(* IEC 61131-3 sources: pub-control-lib/src/02_PubControl, 4 files *)

(* ---- Types.st ---- *)
NAMESPACE Siemens.PubControl.Types
    TYPE
        TankStatus : INT (ACTIVE := 0,  Tapped := 1, TANKING := 2, EMPTY := 4, SERVICE := 3) := ACTIVE;
    END_TYPE

    TYPE
        QualityData : STRUCT
            /// Time how long is tank full with medium (in days)
            occupancyPeriod : REAL;
            /// Time how long tank is empty (in days)
            emptinessPeriod : REAL;
            /// Time how long it needed to empty tank (in days)
            emptyingPeriod : REAL;
            /// delivery date
            deliveryDate : DATE_AND_TIME;
            /// Change inliner last time
            inlinerDate : DATE_AND_TIME;
        END_STRUCT;
    END_TYPE

END_NAMESPACE

(* ---- BasicTapBar.st ---- *)
USING Siemens.PubControl.Interfaces;

NAMESPACE Siemens.PubControl.TapBars
    CLASS BasicTapBar IMPLEMENTS ITapBar
        VAR PRIVATE
            consumption : REAL;
            lastConsumption : REAL;
            flow : REAL;
        END_VAR

        VAR PUBLIC
            WatchDogDiffTime : LTIME;
        END_VAR

        METHOD PUBLIC CalcImpulses
            VAR_INPUT
                MeasureTime : LTIME;
                Impulses : INT;
                Factor : INT;
            END_VAR
            VAR CONSTANT
                HOUR_IN_NS : REAL := REAL#3.6e12;
                ML_IN_L : REAL := REAL#1000.0;
            END_VAR
            VAR_TEMP
                calculatedTime : REAL := REAL#0.0;
            END_VAR
            lastConsumption := (Impulses * Factor)/ML_IN_L;
            consumption := consumption + lastConsumption;

            IF (LTIME#0ns < MeasureTime AND  MeasureTime < WatchDogDiffTime) THEN
                calculatedTime := (TO_REAL(TO_LINT(MeasureTime)));
                flow := lastConsumption * (HOUR_IN_NS/calculatedTime);
            END_IF;
        END_METHOD

        METHOD PUBLIC GetConsumption : REAL
            GetConsumption := consumption;
        END_METHOD

        METHOD PUBLIC GetFlow : REAL
            GetFlow := flow;
        END_METHOD

        METHOD PUBLIC Reset
            consumption := REAL#0.0;
            flow := REAL#0.0;
        END_METHOD

    END_CLASS
END_NAMESPACE

(* ---- TankTap.st ---- *)
USING Siemens.PubControl.Types;
USING Siemens.PubControl.Interfaces;
USING Siemens.PubControl.Types;

NAMESPACE Siemens.PubControl

    // TODO HMI Interface
    CLASS TankTap
        IMPLEMENTS ITank
        VAR PUBLIC
        END_VAR
        VAR PROTECTED
            _maxLevel : UINT;
            _status : TankStatus := TankStatus#ACTIVE;
            _currentLevel : REAL;
            _inTanking : BOOL;
            _inService : BOOL;
        END_VAR

        METHOD PUBLIC SetMaxLevel : INT
            VAR_INPUT
                /// Max level in liter
                MaxLevel : UINT;
            END_VAR
            IF MaxLevel > UINT#0 THEN
                _maxLevel := MaxLevel;
                SetMaxLevel := 0;
            ELSE
                SetMaxLevel := -1;
            END_IF;
            THIS.CheckStatus();
        END_METHOD
        // TODO Test me

        METHOD PUBLIC FINAL Consume : TankStatus
            VAR_INPUT
                /// consumption in liter
                consumption : REAL;
            END_VAR
            IF (_currentLevel - consumption) < 0 THEN
                _currentLevel := 0;
            ELSE
                _currentLevel := _currentLevel - consumption;
            END_IF;
            THIS.CheckStatus();
            Consume := _status;
        END_METHOD
        /// Level in liter

        METHOD PUBLIC GetLevel : UINT
            GetLevel := TO_UINT(_currentLevel);
        END_METHOD

        METHOD PUBLIC GetStatus : TankStatus
            THIS.CheckStatus();
            GetStatus := _status;
        END_METHOD

        METHOD PUBLIC Cleaning
            VAR_INPUT
                Start : BOOL;
                Stop : BOOL;
            END_VAR
            ;
        END_METHOD

        METHOD PROTECTED CheckStatus
            VAR_TEMP
                level : UINT;
            END_VAR
            level := TO_UINT(_currentLevel);
            IF UINT#0 < level AND level < _maxLevel THEN
                _status := TankStatus#TAPPED;
            ELSIF level <= UINT#0 THEN
                _status := TankStatus#EMPTY;
            ELSIF _inTanking THEN
                _status := TankStatus#TANKING;
            ELSIF _inService THEN
                _status := TankStatus#Service;
            ELSE
                _status := TankStatus#ACTIVE;
            END_IF;
        END_METHOD

        METHOD PUBLIC Tanking
            _inTanking := TRUE;
            _currentLevel := _maxLevel;
            _inTanking := FALSE;
        END_METHOD
    END_CLASS

END_NAMESPACE

(* ---- TankWeight.st ---- *)
USING Siemens.PubControl.Interfaces;
USING Siemens.PubControl.Types;

NAMESPACE Siemens.PubControl

    CLASS TankWeight EXTENDS TankTap
        VAR PUBLIC
            /// Weight in kilogram
            Weight : REAL;
        END_VAR
        VAR PROTECTED
            _maxLevelWeight : REAL;
            _factorLevelWeight : REAL;
        END_VAR

        METHOD PUBLIC OVERRIDE SetMaxLevel : INT
            VAR_INPUT
                /// Max level in liter
                MaxLevel : UINT;
            END_VAR
            IF Weight > 0 AND MaxLevel > UINT#0 THEN
                _maxLevel := MaxLevel;
                _currentLevel := MaxLevel;
                _maxLevelWeight := Weight;
                _factorLevelWeight := _maxLevel / _maxLevelWeight;
                SetMaxLevel := 0;
            ELSE
                SetMaxLevel := -1;
            END_IF;
            SUPER.CheckStatus();
        END_METHOD

        /// Level in liter
        METHOD PUBLIC OVERRIDE GetLevel : UINT
            _currentLevel := Weight * _factorLevelWeight;
            SUPER.CheckStatus();
            IF _currentLevel < 0  THEN
                GetLevel := UINT#0;
            ELSE
                GetLevel := TO_UINT(_currentLevel);
            END_IF;

        END_METHOD

    END_CLASS

END_NAMESPACE
